PROGRAM PRG_Test
VAR
	isInRangeFunctionsTest : IsInRangeInclusiveFunctionsTest;
END_VAR

TcUnit.RUN();

END_PROGRAM

(* stored: Version 1.1.0.1, ProductVersion 3.1.4024.15
   POU PRG_Test: Id {1ef4c86c-be7d-46ac-b138-0dab6a048ca7}, SpecialFunc None *)
